PROGRAM P_IncSollRuettel
VAR
END_VAR

IF DB6.iSortierer < 100 THEN
	DB6.iSortierer := DB6.iSortierer + 1;
END_IF

END_PROGRAM

(* stored: Version 1.1.0.1, ProductVersion 3.1.4024.3
   POU P_IncSollRuettel: Id {e574cddf-dcb6-4bd8-939a-53a2adb08fbc}, SpecialFunc None *)
